FUNCTION_BLOCK FB_Raw2Analog_Test extends FB_TestSuite
VAR
END_VAR

TestRawVal2RealValConversion();

METHOD PRIVATE TestRawVal2RealValConversion EXTENDS FB_TestSuite
VAR
	Fb_Raw2Analog	: Fb_AnalogToReal_Conversion;
	nReal : REAL;
	bError : BOOL;
END_VAR
TEST('TestRawVal2RealValConversion');

//Value 1 test
Fb_Raw2Analog(iRawVal:=32676 , iMinVal:=0 , iMaxVal:=100 , lActualVal=> , bError =>bError );
AssertEquals_REAL(	Expected :=100,
					Actual:=Fb_Raw2Analog.lActualVal,
					Delta:= 0.5,
					Message:='Expected Delta < 0.5');

TEST_FINISHED();
END_METHOD

END_FUNCTION_BLOCK

(* stored: Version 1.1.0.1, ProductVersion 3.1.4024.12
   POU FB_Raw2Analog_Test: Id {66030279-90e4-4cb9-bc05-556eb179e71a}, SpecialFunc None
   Method TestRawVal2RealValConversion: Id {67624053-74d8-4f14-acd7-348479c02ac2} *)
